# EPICS autosave request: iocBoot/sioc-sph-im01/sioc-sph-im01.req
file "lcls2toro.req" AREA=SPH,POS=365
